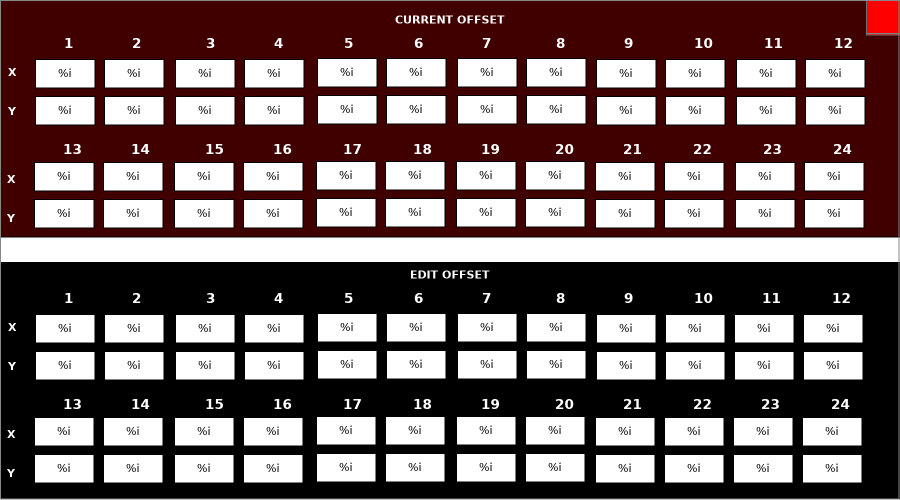
VISUALIZATION MOffset_2  // 900x500
    RoundedRectangle (0,0 900x237)
    Label (0,0 900x40), "CURRENT OFFSET"
    Label (5,55 25x35), "X"
    RoundedRectangle (35,59 60x29), "%i", text variable: Status_GVL.RecipeLine[2].OffsetPattern.Offset_X[1]
    Label (61,26 25x35), "1"
    RoundedRectangle (104,59 60x29), "%i", text variable: Status_GVL.RecipeLine[2].OffsetPattern.Offset_X[2]
    Label (129,26 25x35), "2"
    RoundedRectangle (175,59 60x29), "%i", text variable: Status_GVL.RecipeLine[2].OffsetPattern.Offset_X[3]
    RoundedRectangle (244,59 60x29), "%i", text variable: Status_GVL.RecipeLine[2].OffsetPattern.Offset_X[4]
    Label (5,94 25x35), "Y"
    RoundedRectangle (317,58 60x29), "%i", text variable: Status_GVL.RecipeLine[2].OffsetPattern.Offset_X[5]
    RoundedRectangle (386,58 60x29), "%i", text variable: Status_GVL.RecipeLine[2].OffsetPattern.Offset_X[6]
    RoundedRectangle (457,58 60x29), "%i", text variable: Status_GVL.RecipeLine[2].OffsetPattern.Offset_X[7]
    RoundedRectangle (526,58 60x29), "%i", text variable: Status_GVL.RecipeLine[2].OffsetPattern.Offset_X[8]
    RoundedRectangle (596,59 60x29), "%i", text variable: Status_GVL.RecipeLine[2].OffsetPattern.Offset_X[9]
    RoundedRectangle (665,59 60x29), "%i", text variable: Status_GVL.RecipeLine[2].OffsetPattern.Offset_X[10]
    Label (203,26 25x35), "3"
    Label (271,26 25x35), "4"
    Label (341,26 25x35), "5"
    Label (411,26 25x35), "6"
    Label (479,26 25x35), "7"
    Label (553,26 25x35), "8"
    Label (621,26 25x35), "9"
    Label (691,26 25x35), "10"
    RoundedRectangle (35,96 60x29), "%i", text variable: Status_GVL.RecipeLine[2].OffsetPattern.Offset_Y[1]
    RoundedRectangle (104,96 60x29), "%i", text variable: Status_GVL.RecipeLine[2].OffsetPattern.Offset_Y[2]
    RoundedRectangle (175,96 60x29), "%i", text variable: Status_GVL.RecipeLine[2].OffsetPattern.Offset_Y[3]
    RoundedRectangle (244,96 60x29), "%i", text variable: Status_GVL.RecipeLine[2].OffsetPattern.Offset_Y[4]
    RoundedRectangle (317,95 60x29), "%i", text variable: Status_GVL.RecipeLine[2].OffsetPattern.Offset_Y[5]
    RoundedRectangle (386,95 60x29), "%i", text variable: Status_GVL.RecipeLine[2].OffsetPattern.Offset_Y[6]
    RoundedRectangle (457,95 60x29), "%i", text variable: Status_GVL.RecipeLine[2].OffsetPattern.Offset_Y[7]
    RoundedRectangle (526,95 60x29), "%i", text variable: Status_GVL.RecipeLine[2].OffsetPattern.Offset_Y[8]
    RoundedRectangle (596,96 60x29), "%i", text variable: Status_GVL.RecipeLine[2].OffsetPattern.Offset_Y[9]
    RoundedRectangle (665,96 60x29), "%i", text variable: Status_GVL.RecipeLine[2].OffsetPattern.Offset_Y[10]
    Label (4,162 25x35), "X"
    RoundedRectangle (34,162 60x29), "%i", text variable: Status_GVL.RecipeLine[2].OffsetPattern.Offset_X[13]
    RoundedRectangle (103,162 60x29), "%i", text variable: Status_GVL.RecipeLine[2].OffsetPattern.Offset_X[14]
    RoundedRectangle (174,162 60x29), "%i", text variable: Status_GVL.RecipeLine[2].OffsetPattern.Offset_X[15]
    RoundedRectangle (243,162 60x29), "%i", text variable: Status_GVL.RecipeLine[2].OffsetPattern.Offset_X[16]
    Label (4,201 25x35), "Y"
    RoundedRectangle (316,161 60x29), "%i", text variable: Status_GVL.RecipeLine[2].OffsetPattern.Offset_X[17]
    RoundedRectangle (385,161 60x29), "%i", text variable: Status_GVL.RecipeLine[2].OffsetPattern.Offset_X[18]
    RoundedRectangle (456,161 60x29), "%i", text variable: Status_GVL.RecipeLine[2].OffsetPattern.Offset_X[19]
    RoundedRectangle (525,161 60x29), "%i", text variable: Status_GVL.RecipeLine[2].OffsetPattern.Offset_X[20]
    RoundedRectangle (595,162 60x29), "%i", text variable: Status_GVL.RecipeLine[2].OffsetPattern.Offset_X[21]
    RoundedRectangle (664,162 60x29), "%i", text variable: Status_GVL.RecipeLine[2].OffsetPattern.Offset_X[22]
    RoundedRectangle (34,199 60x29), "%i", text variable: Status_GVL.RecipeLine[2].OffsetPattern.Offset_Y[13]
    RoundedRectangle (103,199 60x29), "%i", text variable: Status_GVL.RecipeLine[2].OffsetPattern.Offset_Y[14]
    RoundedRectangle (174,199 60x29), "%i", text variable: Status_GVL.RecipeLine[2].OffsetPattern.Offset_Y[15]
    RoundedRectangle (243,199 60x29), "%i", text variable: Status_GVL.RecipeLine[2].OffsetPattern.Offset_Y[16]
    RoundedRectangle (316,198 60x29), "%i", text variable: Status_GVL.RecipeLine[2].OffsetPattern.Offset_Y[17]
    RoundedRectangle (385,198 60x29), "%i", text variable: Status_GVL.RecipeLine[2].OffsetPattern.Offset_Y[18]
    RoundedRectangle (456,198 60x29), "%i", text variable: Status_GVL.RecipeLine[2].OffsetPattern.Offset_Y[19]
    RoundedRectangle (525,198 60x29), "%i", text variable: Status_GVL.RecipeLine[2].OffsetPattern.Offset_Y[20]
    RoundedRectangle (595,199 60x29), "%i", text variable: Status_GVL.RecipeLine[2].OffsetPattern.Offset_Y[21]
    RoundedRectangle (664,199 60x29), "%i", text variable: Status_GVL.RecipeLine[2].OffsetPattern.Offset_Y[22]
    Label (60,132 25x35), "13"
    Label (128,132 25x35), "14"
    Label (202,132 25x35), "15"
    Label (270,132 25x35), "16"
    Label (340,132 25x35), "17"
    Label (410,132 25x35), "18"
    Label (478,132 25x35), "19"
    Label (552,132 25x35), "20"
    Label (620,132 25x35), "21"
    Label (690,132 25x35), "22"
    RoundedRectangle (0,262 900x237)
    Label (0,255 900x40), "EDIT OFFSET"
    Label (5,310 25x35), "X"
    RoundedRectangle (35,314 60x29), "%i", text variable: HMI_GVL.arRecipeHMI[2].OffsetPattern.Offset_X[1], input disabled if: Status_GVL.StsEdit[2]
        OnMouseClick: write the text variable via Default
    Label (61,281 25x35), "1"
    RoundedRectangle (104,314 60x29), "%i", text variable: HMI_GVL.arRecipeHMI[2].OffsetPattern.Offset_X[2], input disabled if: Status_GVL.StsEdit[2]
        OnMouseClick: write the text variable via Default
    Label (129,281 25x35), "2"
    RoundedRectangle (175,314 60x29), "%i", text variable: HMI_GVL.arRecipeHMI[2].OffsetPattern.Offset_X[3], input disabled if: Status_GVL.StsEdit[2]
        OnMouseClick: write the text variable via Default
    RoundedRectangle (244,314 60x29), "%i", text variable: HMI_GVL.arRecipeHMI[2].OffsetPattern.Offset_X[4], input disabled if: Status_GVL.StsEdit[2]
        OnMouseClick: write the text variable via Default
    Label (5,349 25x35), "Y"
    RoundedRectangle (317,313 60x29), "%i", text variable: HMI_GVL.arRecipeHMI[2].OffsetPattern.Offset_X[5], input disabled if: Status_GVL.StsEdit[2]
        OnMouseClick: write the text variable via Default
    RoundedRectangle (386,313 60x29), "%i", text variable: HMI_GVL.arRecipeHMI[2].OffsetPattern.Offset_X[6], input disabled if: Status_GVL.StsEdit[2]
        OnMouseClick: write the text variable via Default
    RoundedRectangle (457,313 60x29), "%i", text variable: HMI_GVL.arRecipeHMI[2].OffsetPattern.Offset_X[7], input disabled if: Status_GVL.StsEdit[2]
        OnMouseClick: write the text variable via Default
    RoundedRectangle (526,313 60x29), "%i", text variable: HMI_GVL.arRecipeHMI[2].OffsetPattern.Offset_X[8], input disabled if: Status_GVL.StsEdit[2]
        OnMouseClick: write the text variable via Default
    RoundedRectangle (596,314 60x29), "%i", text variable: HMI_GVL.arRecipeHMI[2].OffsetPattern.Offset_X[9], input disabled if: Status_GVL.StsEdit[2]
        OnMouseClick: write the text variable via Default
    RoundedRectangle (665,314 60x29), "%i", text variable: HMI_GVL.arRecipeHMI[2].OffsetPattern.Offset_X[10], input disabled if: Status_GVL.StsEdit[2]
        OnMouseClick: write the text variable via Default
    Label (203,281 25x35), "3"
    Label (271,281 25x35), "4"
    Label (341,281 25x35), "5"
    Label (411,281 25x35), "6"
    Label (479,281 25x35), "7"
    Label (553,281 25x35), "8"
    Label (621,281 25x35), "9"
    Label (691,281 25x35), "10"
    RoundedRectangle (35,351 60x29), "%i", text variable: HMI_GVL.arRecipeHMI[2].OffsetPattern.Offset_Y[1], input disabled if: Status_GVL.StsEdit[2]
        OnMouseClick: write the text variable via Default
    RoundedRectangle (104,351 60x29), "%i", text variable: HMI_GVL.arRecipeHMI[2].OffsetPattern.Offset_Y[2], input disabled if: Status_GVL.StsEdit[2]
        OnMouseClick: write the text variable via Default
    RoundedRectangle (175,351 60x29), "%i", text variable: HMI_GVL.arRecipeHMI[2].OffsetPattern.Offset_Y[3], input disabled if: Status_GVL.StsEdit[2]
        OnMouseClick: write the text variable via Default
    RoundedRectangle (244,351 60x29), "%i", text variable: HMI_GVL.arRecipeHMI[2].OffsetPattern.Offset_Y[4], input disabled if: Status_GVL.StsEdit[2]
        OnMouseClick: write the text variable via Default
    RoundedRectangle (317,350 60x29), "%i", text variable: HMI_GVL.arRecipeHMI[2].OffsetPattern.Offset_Y[5], input disabled if: Status_GVL.StsEdit[2]
        OnMouseClick: write the text variable via Default
    RoundedRectangle (386,350 60x29), "%i", text variable: HMI_GVL.arRecipeHMI[2].OffsetPattern.Offset_Y[6], input disabled if: Status_GVL.StsEdit[2]
        OnMouseClick: write the text variable via Default
    RoundedRectangle (457,350 60x29), "%i", text variable: HMI_GVL.arRecipeHMI[2].OffsetPattern.Offset_Y[7], input disabled if: Status_GVL.StsEdit[2]
        OnMouseClick: write the text variable via Default
    RoundedRectangle (526,350 60x29), "%i", text variable: HMI_GVL.arRecipeHMI[2].OffsetPattern.Offset_Y[8], input disabled if: Status_GVL.StsEdit[2]
        OnMouseClick: write the text variable via Default
    RoundedRectangle (596,351 60x29), "%i", text variable: HMI_GVL.arRecipeHMI[2].OffsetPattern.Offset_Y[9], input disabled if: Status_GVL.StsEdit[2]
        OnMouseClick: write the text variable via Default
    RoundedRectangle (665,351 60x29), "%i", text variable: HMI_GVL.arRecipeHMI[2].OffsetPattern.Offset_Y[10], input disabled if: Status_GVL.StsEdit[2]
        OnMouseClick: write the text variable via Default
    Label (4,417 25x35), "X"
    RoundedRectangle (34,417 60x29), "%i", text variable: HMI_GVL.arRecipeHMI[2].OffsetPattern.Offset_X[13], input disabled if: Status_GVL.StsEdit[2]
        OnMouseClick: write the text variable via Default
    RoundedRectangle (103,417 60x29), "%i", text variable: HMI_GVL.arRecipeHMI[2].OffsetPattern.Offset_X[14], input disabled if: Status_GVL.StsEdit[2]
        OnMouseClick: write the text variable via Default
    RoundedRectangle (174,417 60x29), "%i", text variable: HMI_GVL.arRecipeHMI[2].OffsetPattern.Offset_X[15], input disabled if: Status_GVL.StsEdit[2]
        OnMouseClick: write the text variable via Default
    RoundedRectangle (243,417 60x29), "%i", text variable: HMI_GVL.arRecipeHMI[2].OffsetPattern.Offset_X[16], input disabled if: Status_GVL.StsEdit[2]
        OnMouseClick: write the text variable via Default
    Label (4,456 25x35), "Y"
    RoundedRectangle (316,416 60x29), "%i", text variable: HMI_GVL.arRecipeHMI[2].OffsetPattern.Offset_X[17], input disabled if: Status_GVL.StsEdit[2]
        OnMouseClick: write the text variable via Default
    RoundedRectangle (385,416 60x29), "%i", text variable: HMI_GVL.arRecipeHMI[2].OffsetPattern.Offset_X[18], input disabled if: Status_GVL.StsEdit[2]
        OnMouseClick: write the text variable via Default
    RoundedRectangle (456,416 60x29), "%i", text variable: HMI_GVL.arRecipeHMI[2].OffsetPattern.Offset_X[19], input disabled if: Status_GVL.StsEdit[2]
        OnMouseClick: write the text variable via Default
    RoundedRectangle (525,416 60x29), "%i", text variable: HMI_GVL.arRecipeHMI[2].OffsetPattern.Offset_X[20], input disabled if: Status_GVL.StsEdit[2]
        OnMouseClick: write the text variable via Default
    RoundedRectangle (595,417 60x29), "%i", text variable: HMI_GVL.arRecipeHMI[2].OffsetPattern.Offset_X[21], input disabled if: Status_GVL.StsEdit[2]
        OnMouseClick: write the text variable via Default
    RoundedRectangle (664,417 60x29), "%i", text variable: HMI_GVL.arRecipeHMI[2].OffsetPattern.Offset_X[22], input disabled if: Status_GVL.StsEdit[2]
        OnMouseClick: write the text variable via Default
    RoundedRectangle (34,454 60x29), "%i", text variable: HMI_GVL.arRecipeHMI[2].OffsetPattern.Offset_Y[13], input disabled if: Status_GVL.StsEdit[2]
        OnMouseClick: write the text variable via Default
    RoundedRectangle (103,454 60x29), "%i", text variable: HMI_GVL.arRecipeHMI[2].OffsetPattern.Offset_Y[14], input disabled if: Status_GVL.StsEdit[2]
        OnMouseClick: write the text variable via Default
    RoundedRectangle (174,454 60x29), "%i", text variable: HMI_GVL.arRecipeHMI[2].OffsetPattern.Offset_Y[15], input disabled if: Status_GVL.StsEdit[2]
        OnMouseClick: write the text variable via Default
    RoundedRectangle (243,454 60x29), "%i", text variable: HMI_GVL.arRecipeHMI[2].OffsetPattern.Offset_Y[16], input disabled if: Status_GVL.StsEdit[2]
        OnMouseClick: write the text variable via Default
    RoundedRectangle (316,453 60x29), "%i", text variable: HMI_GVL.arRecipeHMI[2].OffsetPattern.Offset_Y[17], input disabled if: Status_GVL.StsEdit[2]
        OnMouseClick: write the text variable via Default
    RoundedRectangle (385,453 60x29), "%i", text variable: HMI_GVL.arRecipeHMI[2].OffsetPattern.Offset_Y[18], input disabled if: Status_GVL.StsEdit[2]
        OnMouseClick: write the text variable via Default
    RoundedRectangle (456,453 60x29), "%i", text variable: HMI_GVL.arRecipeHMI[2].OffsetPattern.Offset_Y[19], input disabled if: Status_GVL.StsEdit[2]
        OnMouseClick: write the text variable via Default
    RoundedRectangle (525,453 60x29), "%i", text variable: HMI_GVL.arRecipeHMI[2].OffsetPattern.Offset_Y[20], input disabled if: Status_GVL.StsEdit[2]
        OnMouseClick: write the text variable via Default
    RoundedRectangle (595,454 60x29), "%i", text variable: HMI_GVL.arRecipeHMI[2].OffsetPattern.Offset_Y[21], input disabled if: Status_GVL.StsEdit[2]
        OnMouseClick: write the text variable via Default
    RoundedRectangle (664,454 60x29), "%i", text variable: HMI_GVL.arRecipeHMI[2].OffsetPattern.Offset_Y[22], input disabled if: Status_GVL.StsEdit[2]
        OnMouseClick: write the text variable via Default
    Label (60,387 25x35), "13"
    Label (128,387 25x35), "14"
    Label (202,387 25x35), "15"
    Label (270,387 25x35), "16"
    Label (340,387 25x35), "17"
    Label (410,387 25x35), "18"
    Label (478,387 25x35), "19"
    Label (552,387 25x35), "20"
    Label (620,387 25x35), "21"
    Label (690,387 25x35), "22"
    Button (866,0 35x35), image: VisuSymbols.Symbols.Wrong
        OnMouseClick: CloseDialog Dialog=MOffset_2, Result=OK, NumpadKeypadSet=True
    RoundedRectangle (736,59 60x29), "%i", text variable: Status_GVL.RecipeLine[2].OffsetPattern.Offset_X[11]
    RoundedRectangle (805,59 60x29), "%i", text variable: Status_GVL.RecipeLine[2].OffsetPattern.Offset_X[12]
    Label (761,26 25x35), "11"
    Label (831,26 25x35), "12"
    RoundedRectangle (736,96 60x29), "%i", text variable: Status_GVL.RecipeLine[2].OffsetPattern.Offset_Y[11]
    RoundedRectangle (805,96 60x29), "%i", text variable: Status_GVL.RecipeLine[2].OffsetPattern.Offset_Y[12]
    RoundedRectangle (735,162 60x29), "%i", text variable: Status_GVL.RecipeLine[2].OffsetPattern.Offset_X[23]
    RoundedRectangle (804,162 60x29), "%i", text variable: Status_GVL.RecipeLine[2].OffsetPattern.Offset_X[24]
    RoundedRectangle (735,199 60x29), "%i", text variable: Status_GVL.RecipeLine[2].OffsetPattern.Offset_Y[23]
    RoundedRectangle (804,199 60x29), "%i", text variable: Status_GVL.RecipeLine[2].OffsetPattern.Offset_Y[24]
    Label (760,132 25x35), "23"
    Label (830,132 25x35), "24"
    RoundedRectangle (734,314 60x29), "%i", text variable: HMI_GVL.arRecipeHMI[2].OffsetPattern.Offset_X[11], input disabled if: Status_GVL.StsEdit[2]
        OnMouseClick: write the text variable via Default
    RoundedRectangle (803,314 60x29), "%i", text variable: HMI_GVL.arRecipeHMI[2].OffsetPattern.Offset_X[12], input disabled if: Status_GVL.StsEdit[2]
        OnMouseClick: write the text variable via Default
    Label (759,281 25x35), "11"
    Label (829,281 25x35), "12"
    RoundedRectangle (734,351 60x29), "%i", text variable: HMI_GVL.arRecipeHMI[2].OffsetPattern.Offset_Y[11], input disabled if: Status_GVL.StsEdit[2]
        OnMouseClick: write the text variable via Default
    RoundedRectangle (803,351 60x29), "%i", text variable: HMI_GVL.arRecipeHMI[2].OffsetPattern.Offset_Y[12], input disabled if: Status_GVL.StsEdit[2]
        OnMouseClick: write the text variable via Default
    RoundedRectangle (733,417 60x29), "%i", text variable: HMI_GVL.arRecipeHMI[2].OffsetPattern.Offset_X[23], input disabled if: Status_GVL.StsEdit[2]
        OnMouseClick: write the text variable via Default
    RoundedRectangle (802,417 60x29), "%i", text variable: HMI_GVL.arRecipeHMI[2].OffsetPattern.Offset_X[24], input disabled if: Status_GVL.StsEdit[2]
        OnMouseClick: write the text variable via Default
    RoundedRectangle (733,454 60x29), "%i", text variable: HMI_GVL.arRecipeHMI[2].OffsetPattern.Offset_Y[23], input disabled if: Status_GVL.StsEdit[2]
        OnMouseClick: write the text variable via Default
    RoundedRectangle (802,454 60x29), "%i", text variable: HMI_GVL.arRecipeHMI[2].OffsetPattern.Offset_Y[24], input disabled if: Status_GVL.StsEdit[2]
        OnMouseClick: write the text variable via Default
    Label (758,387 25x35), "23"
    Label (828,387 25x35), "24"
END_VISUALIZATION

(* stored: Version 1.1.0.1, ProductVersion 3.1.4024.12
   Visu MOffset_2: Id {6c952041-ea8a-4190-b6ca-e85e96fb0aca} *)
